PROGRAM PRG_1
VAR
	
	nState: INT;	
	
	bSignalLamp: BOOL;
	
	bSelectorSw: BOOL;
	
	bMotorStart: BOOL;
	bMotorStop: BOOL;
	
	bMotor: BOOL;

	bDelta: BOOL;
	bStar: BOOL;

	bUp: BOOL;
	bDown: BOOL;
	bRight: BOOL;
	bLeft: BOOL;

	bMotorUp: BOOL;
	bMotorDown: BOOL;
	bMotorR: BOOL;
	bMotorL: BOOL;

	bUpSW: BOOL;
	bDownLW: BOOL;
	bRightSW: BOOL;
	bLeftSW: BOOL;
	
	bLedUp: BOOL;
	bLedDown: BOOL;
	bLedR: BOOL;
	bLedL: BOOL;
	
	FlasherRight: FB_Flasher;
	FlasherLeft: FB_Flasher;
	FlasherUp: FB_Flasher;
	FlasherDown: FB_Flasher;
	FB_FlasherCurrency: FB_Flasher;
	FB_FlasherTemp: FB_Flasher;
	
	T1: TON;
	T2: TON;
	
	nValue: INT;
	bFan1: BOOL;
	bFan2: BOOL;
	bTempLamp: BOOL;
	
	
	bEmergecyStop: BOOL;
	bCurrencyLamp: BOOL;
END_VAR



ACT_1();
ACT_3();

IF T2.Q THEN
	
	ACT_2();
			
END_IF



IF bEmergecyStop THEN
	//Her şeyi sıfırla
END_IF

ACTION ACT_1:

T1(IN:=bStar , PT:=T#2M , Q=> , ET=> );
T2(IN:=bMotor , PT:=T#5M , Q=> , ET=> );

CASE nState OF

	0:
	
		IF bSelectorSw THEN
			
			bSignalLamp	:=	TRUE;
			nState := 10;
			FB_FlasherCurrency(bStart:=FALSE);
			
		END_IF
	10:
	
		IF bMotorStart AND NOT bMotorStop THEN
			
			bStar	:=	TRUE;
			bDelta	:= FALSE;
			bMotor	:=	TRUE;
			
			nState := 20;
			
		END_IF
		
	20:	
	
		IF T1.Q THEN
			
			bStar	:=	FALSE;
			bDelta	:= 	TRUE;
			
		END_IF

END_CASE

IF NOT bMotorStart AND bMotorStop	THEN
	
	nState	:=	 0;
	bMotor	:=	FALSE;
	
END_IF

IF T1.Q AND NOT bUp 
AND NOT bDown 
AND NOT bRight
AND NOT bLeft THEN 

	FB_FlasherCurrency(bStart:=TRUE , bLed=>bCurrencyLamp );
	bMotor	:=	FALSE;
	nState	:=	0;
	
END_IF
END_ACTION

ACTION ACT_2:

//LimitSW ler NC olduğu kabul edilmiştir.

FlasherUp(bStart:=bMotorUp , bLed=>bLedUp );
FlasherDown(bStart:=bMotorDown , bLed=>bLedDown );

FlasherRight(bStart:=bMotorR , bLed=>bLedR );
FlasherLeft(bStart:=bMotorL , bLed=>bLedL );


IF bUp AND NOT bDown AND bUpSW THEN
	
	bMotorUp	:=	TRUE;
	bMotorDown	:=	FALSE;	
	
ELSIF bDown AND NOT bUp	AND bDownLW THEN
	
	bMotorUp	:=	FALSE;
	bMotorDown	:=	TRUE;
	
ELSIF	(bDown AND NOT bUp AND NOT bDownLW)
OR		(bUp AND NOT bDown AND NOT bUpSW) 	THEN
		
	bMotorUp	:=	FALSE;
	bMotorDown	:=	FALSE;	
	
END_IF



IF bRight AND NOT bLeft AND bRightSW THEN
	
	bMotorR	:=	TRUE;
	bMotorL	:=	FALSE;


ELSIF NOT bRight AND bLeft AND bLeftSW	THEN
	
	bMotorR	:=	FALSE;
	bMotorL	:=	TRUE;


ELSIF	(bRight	AND NOT bLeft AND NOT bRightSW)
OR 		(bLeft	AND NOT bRight AND NOT bLeftSW) THEN
		
	bMotorR	:=	FALSE;
	bMotorL	:=	FALSE;	
	
END_IF
END_ACTION

ACTION ACT_3:


FB_FlasherTemp(bStart:=bFan2, bLed=>bTempLamp );


IF nValue	>=	10 AND	nValue	<=	20 THEN		// Kademe_1
	
	bFan1	:=	TRUE;
	bFan2	:=	FALSE;
	
ELSIF	nValue > 20 THEN	//	Kademe_2
	
	bFan1	:=	TRUE;
	bFan2	:=	TRUE;
	
	bMotor	:=	FALSE;
	
	nState	:=	0;
	
END_IF
END_ACTION

END_PROGRAM

(* stored: Version 1.1.0.1, ProductVersion 3.1.4024.4
   POU PRG_1: Id {48f4c5fc-9c25-4924-80b2-be75e976656f}, SpecialFunc None
   Action ACT_1: Id {404c97d7-c55a-43ac-9da2-2aa96dc8badf}
   Action ACT_2: Id {6509ad7e-7224-42f9-b593-8ee016e9f99f}
   Action ACT_3: Id {4fe8f9df-61cc-4dd5-931a-bcaa2361f4bf} *)
